// TwinCAT 3 PLC project Untitled1
// ProgramVersion: 3.1.4024.12
// libraries:
//   Tc2_Standard, * (Beckhoff Automation GmbH)
//   Tc2_System, * (Beckhoff Automation GmbH)
//   Tc3_Module, * (Beckhoff Automation GmbH)
// project tree:
//   GVLs/ GVL.TcGVL
//   / PlcTask.TcTTO
//   POUs/ MAIN.TcPOU
// real-time tasks:
//   TASK PlcTask: cycle T#10ms, priority 20, ADS port 350
// I/O:
//   DEVICE Device 1 (EtherCAT), AmsNetId 10.0.0.16.2.1
//     Term 1 (EK1100) [EK1100 EtherCAT Coupler (2A E-Bus)]
//       Term 2 (EL6851) [EL6851 DMX Master]
//       Term 3 (EL1008) [EL1008 8Ch. Dig. Input 24V, 3ms]
//       Term 4 (EL1008) [EL1008 8Ch. Dig. Input 24V, 3ms]
//       Term 5 (EL1008) [EL1008 8Ch. Dig. Input 24V, 3ms]
//       Term 6 (EL1008) [EL1008 8Ch. Dig. Input 24V, 3ms]
//       Term 7 (EL1008) [EL1008 8Ch. Dig. Input 24V, 3ms]
//       Term 8 (EL1008) [EL1008 8Ch. Dig. Input 24V, 3ms]
//       Term 9 (EL1008) [EL1008 8Ch. Dig. Input 24V, 3ms]
//       Term 10 (EL1008) [EL1008 8Ch. Dig. Input 24V, 3ms]
//       Term 11 (EL1008) [EL1008 8Ch. Dig. Input 24V, 3ms]
//       Term 12 (EL1008) [EL1008 8Ch. Dig. Input 24V, 3ms]
//       Term 13 (EL1088) [EL1088 8Ch. Dig. Input 24V, 3ms, negative]
//       Term 14 (EL1088) [EL1088 8Ch. Dig. Input 24V, 3ms, negative]
//       Term 15 (EL1088) [EL1088 8Ch. Dig. Input 24V, 3ms, negative]
//       Term 16 (EL1088) [EL1088 8Ch. Dig. Input 24V, 3ms, negative]
//       Term 17 (EL1088) [EL1088 8Ch. Dig. Input 24V, 3ms, negative]
//       Term 18 (EL9410) [EL9410 E-Bus Power Supplier  (Diagnostics)]
//       Term 19 (EL1088) [EL1088 8Ch. Dig. Input 24V, 3ms, negative]
//       Term 20 (EL1088) [EL1088 8Ch. Dig. Input 24V, 3ms, negative]
//       Term 21 (EL1088) [EL1088 8Ch. Dig. Input 24V, 3ms, negative]
//       Term 22 (EL1088) [EL1088 8Ch. Dig. Input 24V, 3ms, negative]
//       Term 23 (EL1088) [EL1088 8Ch. Dig. Input 24V, 3ms, negative]
//       Term 24 (EL9011) [EL9011 End Terminal]
// variable links:
//   Untitled1/Untitled1 Instance <-> Device 1 (EtherCAT)/Term 1 (EK1100)/Term 10 (EL1008)
//     PlcTask Inputs/MAIN.arrInputPNP[{56..63}] <-> Channel {1..8}/Input  (8 links)
//   Untitled1/Untitled1 Instance <-> Device 1 (EtherCAT)/Term 1 (EK1100)/Term 11 (EL1008)
//     PlcTask Inputs/MAIN.arrInputPNP[{64..71}] <-> Channel {1..8}/Input  (8 links)
//   Untitled1/Untitled1 Instance <-> Device 1 (EtherCAT)/Term 1 (EK1100)/Term 12 (EL1008)
//     PlcTask Inputs/MAIN.arrInputPNP[{72..79}] <-> Channel {1..8}/Input  (8 links)
//   Untitled1/Untitled1 Instance <-> Device 1 (EtherCAT)/Term 1 (EK1100)/Term 13 (EL1088)
//     PlcTask Inputs/MAIN.arrInputNPN[{0..7}] <-> Channel {1..8}/Input  (8 links)
//   Untitled1/Untitled1 Instance <-> Device 1 (EtherCAT)/Term 1 (EK1100)/Term 14 (EL1088)
//     PlcTask Inputs/MAIN.arrInputNPN[{8..15}] <-> Channel {1..8}/Input  (8 links)
//   Untitled1/Untitled1 Instance <-> Device 1 (EtherCAT)/Term 1 (EK1100)/Term 15 (EL1088)
//     PlcTask Inputs/MAIN.arrInputNPN[{16..23}] <-> Channel {1..8}/Input  (8 links)
//   Untitled1/Untitled1 Instance <-> Device 1 (EtherCAT)/Term 1 (EK1100)/Term 16 (EL1088)
//     PlcTask Inputs/MAIN.arrInputNPN[{24..31}] <-> Channel {1..8}/Input  (8 links)
//   Untitled1/Untitled1 Instance <-> Device 1 (EtherCAT)/Term 1 (EK1100)/Term 17 (EL1088)
//     PlcTask Inputs/MAIN.arrInputNPN[{32..39}] <-> Channel {1..8}/Input  (8 links)
//   Untitled1/Untitled1 Instance <-> Device 1 (EtherCAT)/Term 1 (EK1100)/Term 19 (EL1088)
//     PlcTask Inputs/MAIN.arrInputNPN[{40..47}] <-> Channel {1..8}/Input  (8 links)
//   Untitled1/Untitled1 Instance <-> Device 1 (EtherCAT)/Term 1 (EK1100)/Term 20 (EL1088)
//     PlcTask Inputs/MAIN.arrInputNPN[{48..55}] <-> Channel {1..8}/Input  (8 links)
//   Untitled1/Untitled1 Instance <-> Device 1 (EtherCAT)/Term 1 (EK1100)/Term 21 (EL1088)
//     PlcTask Inputs/MAIN.arrInputNPN[{56..63}] <-> Channel {1..8}/Input  (8 links)
//   Untitled1/Untitled1 Instance <-> Device 1 (EtherCAT)/Term 1 (EK1100)/Term 22 (EL1088)
//     PlcTask Inputs/MAIN.arrInputNPN[{64..71}] <-> Channel {1..8}/Input  (8 links)
//   Untitled1/Untitled1 Instance <-> Device 1 (EtherCAT)/Term 1 (EK1100)/Term 23 (EL1088)
//     PlcTask Inputs/MAIN.arrInputNPN[{72..79}] <-> Channel {1..8}/Input  (8 links)
//   Untitled1/Untitled1 Instance <-> Device 1 (EtherCAT)/Term 1 (EK1100)/Term 3 (EL1008)
//     PlcTask Inputs/MAIN.arrInputPNP[{0..7}] <-> Channel {1..8}/Input  (8 links)
//   Untitled1/Untitled1 Instance <-> Device 1 (EtherCAT)/Term 1 (EK1100)/Term 4 (EL1008)
//     PlcTask Inputs/MAIN.arrInputPNP[{8..15}] <-> Channel {1..8}/Input  (8 links)
//   Untitled1/Untitled1 Instance <-> Device 1 (EtherCAT)/Term 1 (EK1100)/Term 5 (EL1008)
//     PlcTask Inputs/MAIN.arrInputPNP[{16..23}] <-> Channel {1..8}/Input  (8 links)
//   Untitled1/Untitled1 Instance <-> Device 1 (EtherCAT)/Term 1 (EK1100)/Term 6 (EL1008)
//     PlcTask Inputs/MAIN.arrInputPNP[{24..31}] <-> Channel {1..8}/Input  (8 links)
//   Untitled1/Untitled1 Instance <-> Device 1 (EtherCAT)/Term 1 (EK1100)/Term 7 (EL1008)
//     PlcTask Inputs/MAIN.arrInputPNP[{32..39}] <-> Channel {1..8}/Input  (8 links)
//   Untitled1/Untitled1 Instance <-> Device 1 (EtherCAT)/Term 1 (EK1100)/Term 8 (EL1008)
//     PlcTask Inputs/MAIN.arrInputPNP[{40..47}] <-> Channel {1..8}/Input  (8 links)
//   Untitled1/Untitled1 Instance <-> Device 1 (EtherCAT)/Term 1 (EK1100)/Term 9 (EL1008)
//     PlcTask Inputs/MAIN.arrInputPNP[{48..55}] <-> Channel {1..8}/Input  (8 links)

CONFIGURATION Untitled1
    RESOURCE PLC ON TwinCAT3
        TASK PlcTask(INTERVAL := T#10ms, PRIORITY := 20);
        PROGRAM MAIN WITH PlcTask : MAIN;
    END_RESOURCE
END_CONFIGURATION

// ---- GVLs/GVL.TcGVL
{attribute 'qualified_only'}
VAR_GLOBAL CONSTANT
	cuiNrChannel		: UINT	:= 79;
END_VAR

// ---- POUs/MAIN.TcPOU
PROGRAM MAIN
VAR
	arrInputPNP AT %I* : ARRAY[0..GVL.cuiNrChannel] OF BOOL;
	arrInputNPN	AT %I* : ARRAY[0..GVL.cuiNrChannel] OF BOOL;
END_VAR

arrInputPNP;
arrInputNPN;

END_PROGRAM
